FUNCTION F_SettingItemHandlingWs : WSTRING
VAR_IN_OUT
	wsValue		: WSTRING;
	stSetting 	: ST_Data_Item;
END_VAR
VAR
	stInfo 		: ST_Text;
	sChanges	: T_MaxString;
	IEvent		: I_EventHandler;
END_VAR

F_SettingItemHandlingWs := stSetting.sValue;

IF Services.bSettingsSaved OR NOT Services.bPlcInitDone THEN
	wsValue := stSetting.sValue;
	RETURN;
END_IF

IF wsValue = stSetting.sValue THEN
	RETURN;
END_IF

sChanges := sEmpty;
IEvent := Services.fbEventHandler;

// 1. chk user level
IF NOT F_ChkSettingUserLevel(HMI.eUserLevel, stSetting, stInfo => stInfo) THEN							  
	IEvent.Select(TC_Events.SettingsEventClass.WarningEvent)
		  .ArgAddWString(stInfo.wsName)
		  .Raise();
							
	wsValue := stSetting.sValue;
	RETURN;
END_IF


// 2. chk min/max value
//IF NOT F_ChkSettingLimitF(wsValue, stSetting, stInfo => stInfo) THEN
//	IEvent.Select(TC_Events.SettingsEventClass.WarningEvent)
//		  .ArgAddWString(stInfo.wsName)
//		  .Raise();
//							
//	wsValue := stSetting.sValue;
//	RETURN;
//END_IF

// 3. save changes

IF stSetting.eDataType = E_DataType.eDataType_wstring THEN
	F_TrackSettingChangesWs(wsValue, stSetting, sChanges);
END_IF

// 4. track settings changes
IF sChanges <> sEmpty THEN
	ILog.AddLog(Concat5('Settings Changed, ', 'EKS level: ', TO_STRING(HMI.eUserLevel), '. Changes: ', sChanges), 
				'HMI Controller', 
				E_LogLevel.eLogLevel_info);
END_IF

wsValue := stSetting.sValue;
F_SettingItemHandlingWs := stSetting.sValue;

END_FUNCTION

(* stored: Version 1.1.0.1
   POU F_SettingItemHandlingWs: Id {c1beea03-d786-4e8f-a6ed-1dceacf26744}, SpecialFunc None *)
